TYPE Read_BLPS3_Values_To_PC_Struct :
UNION
	S_BLPS3Values_To_PC:S_BLPS3Values_To_PC_Struct;
END_UNION
END_TYPE

(* stored: Version 1.1.0.1, ProductVersion 3.1.4024.16
   DUT Read_BLPS3_Values_To_PC_Struct: Id {a2be2012-8d99-41ef-a65c-2785bc94003f} *)
